// TIA Portal V17 export
// export: Created 2025-03-05T08:03:48.0833325Z, ExportSetting WithDefaults, DisplayName Totally Integrated Automation Portal, DisplayVersion V17 Update 8, DisplayName TIA Portal Openness, DisplayVersion V17 Update 8, DisplayName TIA Portal Version Control Interface, DisplayVersion V17, DisplayName SINAMICS Startdrive Advanced, DisplayVersion V17 SP2, DisplayName SINAMICS Startdrive G110M, G120, G120C, G120D, G120P, G115D, DisplayVersion V17 SP2, DisplayName SINAMICS Startdrive G130, G150, S120, S150, SINAMICS MV, S210, DisplayVersion V17 SP2, DisplayName STEP 7 Professional, DisplayVersion V17 Update 8, DisplayName SINUMERIK ONE STEP 7 Toolbox, DisplayVersion V17 Update 12, DisplayName SINUMERIK 840D sl STEP 7 Toolbox, DisplayVersion V17 Update 12, DisplayName STEP 7 Safety, DisplayVersion V17 Update 6, DisplayName WinCC Advanced, DisplayVersion V17 Update 8
TYPE "WINCC_HMI_LINES"
// stored: IsFailsafeCompliant false
   STRUCT
      WINCC_LINE_REQUEST_RIGHT : Bool;   // RIGHT REQUEST
      WINCC_LINE_REQUEST_LEFT : Bool;   // LEFT REQUEST
      WINCC_LINE_CONDITIONS_RIGHT : Bool;   // RIGHT CONDITIONS
      WINCC_LINE_CONDITIONS_LEFT : Bool;   // LEFT CONDITIONS
      WINCC_LINE_ACTIVE_RIGHT : Bool;   // RIGHT ACTIVE
      WINCC_LINE_ACTIVE_LEFT : Bool;   // LEFT ACTIVE
      WINCC_LINE_STATUS_1_RIGHT : Bool;   // RIGHT STATUS 1
      WINCC_LINE_STATUS_1_LEFT : Bool;   // LEFT STATUS 1
      WINCC_LINE_STATUS_2_RIGHT : Bool;   // RIGHT STATUS 2
      WINCC_LINE_STATUS_2_LEFT : Bool;   // LEFT STATUS 2
      WINCC_LINE_STATUS_3_RIGHT : Bool;   // RIGHT STATUS 3
      WINCC_LINE_STATUS_3_LEFT : Bool;   // LEFT STATUS 3
      WINCC_LINE_STATUS_4_RIGHT : Bool;   // RIGHT STATUS 4
      WINCC_LINE_STATUS_4_LEFT : Bool;   // LEFT STATUS 4
      WINCC_LINE_STATUS_5_RIGHT : Bool;   // RIGHT STATUS 5
      WINCC_LINE_STATUS_5_LEFT : Bool;   // LEFT STATUS 5
   END_STRUCT;
END_TYPE
